{attribute 'qualified_only'}
{attribute 'strict'}
TYPE E_Gamepad_Handshake_State :
(
	// No handshake attempt has run yet
	NotStarted := 0,
	// The read of the service info block is in flight
	Busy := 1,
	// The service answered and the contract versions are compatible
	Compatible := 2,
	// The last attempt got no answer. The service predates the info block or was not
	// reachable yet; the handshake keeps retrying. Data exchange still works
	Unsupported := 3,
	// The service speaks a newer contract major version. Check for a library update
	Mismatch := 4
);
END_TYPE

(* stored: Version 1.1.0.1, ProductVersion 3.1.4024.11
   DUT E_Gamepad_Handshake_State: Id {a599cfcb-e618-4094-8186-3c7659e4937e} *)
